TYPE ST_AxisMapping :
STRUCT
	name : STRING;
	indexOffset : UDINT;
	pAny : MPM_JsonParser.ST_AnyType_User;
END_STRUCT
END_TYPE

(* stored: Version 1.1.0.1, ProductVersion 3.1.4024.12
   DUT ST_AxisMapping: Id {efcb00d1-0caa-4cae-abd7-242813a416c4} *)
